{attribute 'linkalways'} 
{attribute 'no_explicit_call' := 'This FB is a CLASS and must be accessed using methods or properties'}
{attribute 'enable_dynamic_creation'}
FUNCTION_BLOCK _STRING EXTENDS DatatypeBase
VAR
	localData : T_MaxString;
	activeData : REFERENCE TO T_MaxString REF= localData;
END_VAR

PROPERTY PUBLIC Address : PVOID
GET
Address := ADR(activeData);
END_GET
END_PROPERTY

METHOD PUBLIC ClearReference
VAR_INPUT
END_VAR
activeData REF= localData;
END_METHOD

METHOD PUBLIC Clone : I_Datatype
VAR
    pClone : POINTER TO _STRING;
END_VAR
pClone := __NEW(_STRING(InitialValue := Value));
Clone := pClone^;
END_METHOD

METHOD FB_init : BOOL
VAR_INPUT
	bInitRetains : BOOL; // if TRUE, the retain variables are initialized (warm start / cold start)
	bInCopyCode : BOOL;  // if TRUE, the instance afterwards gets moved WORDo the copy code (online change)
	InitialValue : T_MaxString;
END_VAR
localData := InitialValue;
END_METHOD

METHOD PUBLIC MakeReferenceTo
VAR_INPUT
	ReferenceTarget : REFERENCE TO T_MaxString;
END_VAR
activeData REF= ReferenceTarget;
END_METHOD

METHOD PUBLIC SerializeWith
VAR_INPUT
	Serializer : I_Serializer;
END_VAR
Serializer.AddString(activeData);
END_METHOD

PROPERTY PUBLIC Size : UDINT
GET
Size := SIZEOF(activeData);
END_GET
END_PROPERTY

METHOD TryDeserializeFrom : BOOL
VAR_INPUT
	Deserializer : I_Deserializer;
	Feedback : I_DeserializerFeedback;
END_VAR
TryDeserializeFrom := Deserializer.TryGetString(activeData, Feedback);
END_METHOD

METHOD TryMakeReferenceTo : BOOL
VAR_INPUT
	Target : I_Datatype;
END_VAR
VAR
	pTargetData : POINTER TO T_MaxString;
END_VAR
IF NOT (Target.TypeName = TypeName) THEN
	RETURN;
END_IF

pTargetData := Target.Address;
activeData REF= pTargetData^;
TryMakeReferenceTo := TRUE;
END_METHOD

PROPERTY PUBLIC TypeName : T_MAXSTRING
GET
TypeName := 'STRING';
END_GET
END_PROPERTY

PROPERTY PUBLIC Value : T_MaxString
GET
Value := activeData;
END_GET
SET
activeData := Value;
END_SET
END_PROPERTY

END_FUNCTION_BLOCK

(* stored: Version 1.1.0.1, ProductVersion 3.1.4024.12
   POU _STRING: Id {e34be6f6-ed11-4620-954b-fc59662a1046}, SpecialFunc None
   Folder Constructor: Id {dd58c89a-155d-4574-b6af-e4353333780b}
   Property Address: Id {63cfd837-ca02-42ac-a331-b6a79dc69cba}
   Get Get: Id {48e4edf2-3b35-463a-a0a0-fdb358543548}
   Method ClearReference: Id {748f1968-4e1a-4626-9f38-f6709e4e2c8c}
   Method Clone: Id {d34f0c28-9732-495b-af1a-52f63da75e91}
   Method FB_init: Id {37120b81-68ce-4c13-b9f5-e936732b021d}
   Method MakeReferenceTo: Id {7f64c2c2-3c77-47ea-bd28-1b5bb5b0e2b0}
   Method SerializeWith: Id {85b11fb1-ef00-468d-9302-51a27f94c10b}
   Property Size: Id {cbf10651-cbd3-4204-9c43-c4e897fd0649}
   Get Get: Id {9549af45-4750-421b-8006-69e5d1807263}
   Method TryDeserializeFrom: Id {263d0a40-070b-4131-8b48-06f2a957fe3e}
   Method TryMakeReferenceTo: Id {10c93950-7080-4e3b-ba07-f647051f1cd5}
   Property TypeName: Id {f6b5bec0-9ee7-423e-8fe7-575682b38629}
   Get Get: Id {4555024a-3ef5-4237-8e0d-aa7bcb6a98fe}
   Property Value: Id {2361cef7-08a2-4885-b0fa-340048a39919}
   Get Get: Id {cced6fc2-1a7e-41ad-b632-fccbc4510b25}
   Set Set: Id {7e0501ed-f25e-4954-866b-0925d0671d01} *)
